PROGRAM MAIN
VAR
	{IF defined (TestVariant1)}
	sVariantName 	: STRING := 'TestVariant1';
	{ELSE}
	sVariantName	: STRING := 'TestVariant2';
	{END_IF}
END_VAR

END_PROGRAM

(* stored: Version 1.1.0.1, ProductVersion 3.1.4024.3
   POU MAIN: Id {e1a68a50-22b2-4ff7-bc63-b3e286c69b24}, SpecialFunc None *)
